// TIA Portal V17 export
// export: Created 2024-01-13T10:15:25.0475265Z, ExportSetting WithDefaults, DisplayName Totally Integrated Automation Portal, DisplayVersion V17, DisplayName TIA Portal Openness, DisplayVersion V17, DisplayName TIA Portal Version Control Interface, DisplayVersion V17, DisplayName STEP 7 Professional, DisplayVersion V17, DisplayName STEP 7 Safety, DisplayVersion V17, DisplayName WinCC Advanced, DisplayVersion V17
FUNCTION "9.1 ACCS Crane Number" : Void   // FC25, LAD
TITLE = Change ACCS Crane ID to Crane ID for Check
{ S7_Optimized_Access := 'TRUE' }
VERSION : 0.1
// stored: AutoNumber false, IsIECCheckEnabled false, SetENOAutomatically false, UDAEnableTagReadback false
   VAR_INPUT
      crane_number : Int;
   END_VAR
   VAR_OUTPUT
      CraneID : Int;
   END_VAR
BEGIN

REGION Network 1: 102
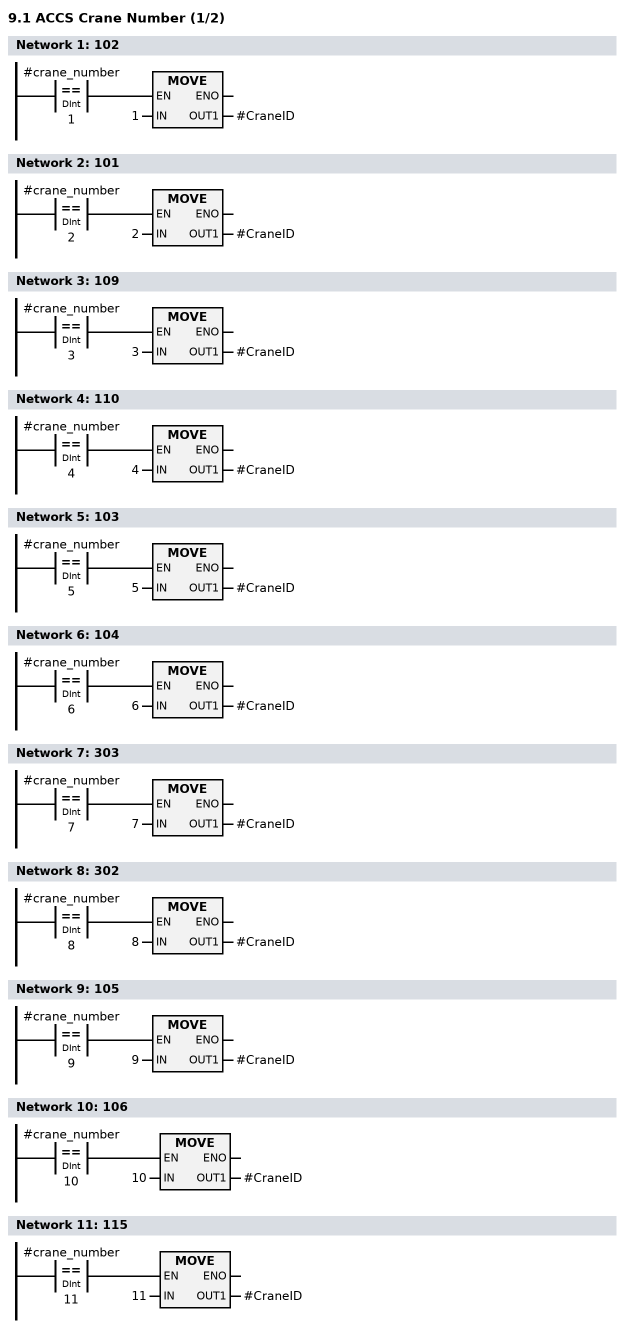
   RUNG wire#powerrail
      { S7_Templates := "SrcType := DInt" } EQ_Contact(in1 := #crane_number, in2 := 1)
      Move(in := 1, out1 => #CraneID)
   END_RUNG
   // the same network as SCL:
   IF #crane_number = 1 THEN #CraneID := 1; END_IF;
END_REGION

REGION Network 2: 101
   RUNG wire#powerrail
      { S7_Templates := "SrcType := DInt" } EQ_Contact(in1 := #crane_number, in2 := 2)
      Move(in := 2, out1 => #CraneID)
   END_RUNG
   // the same network as SCL:
   IF #crane_number = 2 THEN #CraneID := 2; END_IF;
END_REGION

REGION Network 3: 109
   RUNG wire#powerrail
      { S7_Templates := "SrcType := DInt" } EQ_Contact(in1 := #crane_number, in2 := 3)
      Move(in := 3, out1 => #CraneID)
   END_RUNG
   // the same network as SCL:
   IF #crane_number = 3 THEN #CraneID := 3; END_IF;
END_REGION

REGION Network 4: 110
   RUNG wire#powerrail
      { S7_Templates := "SrcType := DInt" } EQ_Contact(in1 := #crane_number, in2 := 4)
      Move(in := 4, out1 => #CraneID)
   END_RUNG
   // the same network as SCL:
   IF #crane_number = 4 THEN #CraneID := 4; END_IF;
END_REGION

REGION Network 5: 103
   RUNG wire#powerrail
      { S7_Templates := "SrcType := DInt" } EQ_Contact(in1 := #crane_number, in2 := 5)
      Move(in := 5, out1 => #CraneID)
   END_RUNG
   // the same network as SCL:
   IF #crane_number = 5 THEN #CraneID := 5; END_IF;
END_REGION

REGION Network 6: 104
   RUNG wire#powerrail
      { S7_Templates := "SrcType := DInt" } EQ_Contact(in1 := #crane_number, in2 := 6)
      Move(in := 6, out1 => #CraneID)
   END_RUNG
   // the same network as SCL:
   IF #crane_number = 6 THEN #CraneID := 6; END_IF;
END_REGION

REGION Network 7: 303
   RUNG wire#powerrail
      { S7_Templates := "SrcType := DInt" } EQ_Contact(in1 := #crane_number, in2 := 7)
      Move(in := 7, out1 => #CraneID)
   END_RUNG
   // the same network as SCL:
   IF #crane_number = 7 THEN #CraneID := 7; END_IF;
END_REGION

REGION Network 8: 302
   RUNG wire#powerrail
      { S7_Templates := "SrcType := DInt" } EQ_Contact(in1 := #crane_number, in2 := 8)
      Move(in := 8, out1 => #CraneID)
   END_RUNG
   // the same network as SCL:
   IF #crane_number = 8 THEN #CraneID := 8; END_IF;
END_REGION

REGION Network 9: 105
   RUNG wire#powerrail
      { S7_Templates := "SrcType := DInt" } EQ_Contact(in1 := #crane_number, in2 := 9)
      Move(in := 9, out1 => #CraneID)
   END_RUNG
   // the same network as SCL:
   IF #crane_number = 9 THEN #CraneID := 9; END_IF;
END_REGION

REGION Network 10: 106
   RUNG wire#powerrail
      { S7_Templates := "SrcType := DInt" } EQ_Contact(in1 := #crane_number, in2 := 10)
      Move(in := 10, out1 => #CraneID)
   END_RUNG
   // the same network as SCL:
   IF #crane_number = 10 THEN #CraneID := 10; END_IF;
END_REGION

REGION Network 11: 115
   RUNG wire#powerrail
      { S7_Templates := "SrcType := DInt" } EQ_Contact(in1 := #crane_number, in2 := 11)
      Move(in := 11, out1 => #CraneID)
   END_RUNG
   // the same network as SCL:
   IF #crane_number = 11 THEN #CraneID := 11; END_IF;
END_REGION

REGION Network 12: 116
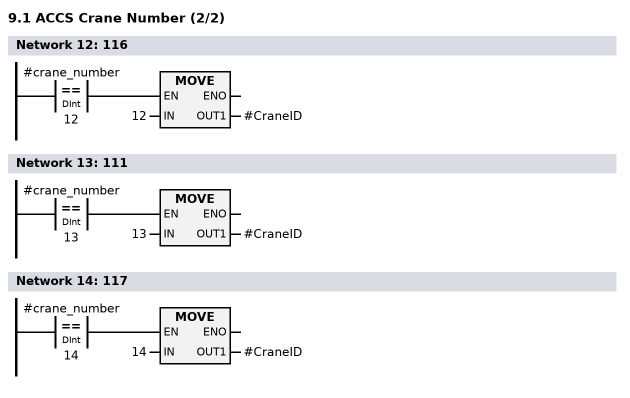
   RUNG wire#powerrail
      { S7_Templates := "SrcType := DInt" } EQ_Contact(in1 := #crane_number, in2 := 12)
      Move(in := 12, out1 => #CraneID)
   END_RUNG
   // the same network as SCL:
   IF #crane_number = 12 THEN #CraneID := 12; END_IF;
END_REGION

REGION Network 13: 111
   RUNG wire#powerrail
      { S7_Templates := "SrcType := DInt" } EQ_Contact(in1 := #crane_number, in2 := 13)
      Move(in := 13, out1 => #CraneID)
   END_RUNG
   // the same network as SCL:
   IF #crane_number = 13 THEN #CraneID := 13; END_IF;
END_REGION

REGION Network 14: 117
   RUNG wire#powerrail
      { S7_Templates := "SrcType := DInt" } EQ_Contact(in1 := #crane_number, in2 := 14)
      Move(in := 14, out1 => #CraneID)
   END_RUNG
   // the same network as SCL:
   IF #crane_number = 14 THEN #CraneID := 14; END_IF;
END_REGION
END_FUNCTION
